{attribute 'qualified_only'}
VAR_GLOBAL
	CoffeeReady: BOOL := FALSE;

	CLEANING: BOOL := FALSE;

	Message: STRING;
	Tclean: Ton;
END_VAR

(* stored: Version 1.1.0.1, ProductVersion 3.1.4024.15
   GVL GVL: Id {7c99cd67-5fc7-4eb9-9e45-cac69ab510bd} *)
